{attribute 'linkalways'} 
{attribute 'no_explicit_call' := 'This FB is a CLASS and must be accessed using methods or properties'}
{attribute 'enable_dynamic_creation'}
FUNCTION_BLOCK ABSTRACT AliasDatatypeBase EXTENDS UserDefinedDatatypeBase IMPLEMENTS I_AliasDatatype
VAR
	_baseDatatype : I_Datatype;
END_VAR

METHOD PROTECTED AddBaseDatatype
VAR_INPUT
	BaseType : I_Datatype;
END_VAR
_baseDatatype := BaseType;
END_METHOD

PROPERTY PUBLIC BaseDatatype : I_Datatype
GET
BaseDatatype := _baseDatatype;
END_GET
END_PROPERTY

METHOD PROTECTED OnSerializeTypeWith
VAR_INPUT
	Serializer : I_Serializer;
END_VAR
SUPER^.OnSerializeTypeWith(Serializer);
Serializer.AddKey('baseDatatype');
_baseDatatype.SerializeTypeWith(Serializer);
END_METHOD

METHOD PUBLIC SerializeWith
VAR_INPUT
	Serializer : I_Serializer;
END_VAR
_baseDatatype.SerializeWith(Serializer);
END_METHOD

METHOD TryDeserializeFrom : BOOL
VAR_INPUT
	Deserializer : I_Deserializer;
	Feedback : I_DeserializerFeedback;
END_VAR
TryDeserializeFrom := _baseDatatype.TryDeserializeFrom(Deserializer, Feedback);
END_METHOD

METHOD PUBLIC TryResolveAsAliasDatatype : BOOL
VAR_INPUT
	Destination : REFERENCE TO I_AliasDatatype;
END_VAR
Destination := THIS^;
TryResolveAsAliasDatatype := TRUE;
END_METHOD

PROPERTY PUBLIC TypeName : T_MAXSTRING
GET
TypeName := 'ALIAS';
END_GET
END_PROPERTY

END_FUNCTION_BLOCK

(* stored: Version 1.1.0.1, ProductVersion 3.1.4024.12
   POU AliasDatatypeBase: Id {eb83021a-1b0f-06f6-18a4-df8e0c17d29e}, SpecialFunc None
   Folder Protected: Id {234fb5d9-3841-00d9-21c3-acc7d986e743}
   Method AddBaseDatatype: Id {b0561277-6f84-0cd1-3be8-7def729ba8f8}
   Property BaseDatatype: Id {9c84384a-fdb6-0d72-2583-e69351dfb7eb}
   Get Get: Id {2b819f6f-3935-00de-379f-3e611f19b398}
   Method OnSerializeTypeWith: Id {f846069a-b6a1-0199-3b45-e4c9efc89bac}
   Method SerializeWith: Id {c906ad78-238b-01cc-0797-6b811d9bfb45}
   Method TryDeserializeFrom: Id {2b54a508-d98b-01d3-04be-6db794e7b76b}
   Method TryResolveAsAliasDatatype: Id {789b9163-85fd-0a42-1794-faeaaf2c520d}
   Property TypeName: Id {5f086b0e-0db7-04c0-1b39-f1e395459705}
   Get Get: Id {67d55b3b-3b4d-03a8-3932-8e8f14bf44a4} *)
